// TIA Portal V17 export
// export: Created 2024-08-09T12:53:13.8222628Z, ExportSetting WithDefaults, DisplayName Totally Integrated Automation Portal, DisplayVersion V17 Update 7, DisplayName TIA Portal Openness, DisplayVersion V17 Update 7, DisplayName TIA Portal Version Control Interface, DisplayVersion V17, DisplayName STEP 7 Professional, DisplayVersion V17 Update 7, DisplayName STEP 7 Safety, DisplayVersion V17 Update 6, DisplayName WinCC Professional, DisplayVersion V17 Update 7
VAR_GLOBAL   // PLC tag table "TREMIE_TRAPPE"
END_VAR
VAR_GLOBAL CONSTANT   // user constants
   NIV_TREMIE_TRAPPE_DEBUT_LOT : USInt := 1;
   NIV_TREMIE_TRAPPE_AUT_REMP : USInt := 10;
   NIV_TREMIE_TRAPPE_PRES_PRD : USInt := 20;
   NIV_TREMIE_TRAPPE_ATT_FIN_TROU : USInt := 25;
   NIV_TREMIE_TRAPPE_DEM_EXTRACT : USInt := 30;
   NIV_TREMIE_TRAPPE_NB : USInt := 45;
   NIV_TREMIE_TRAPPE_VID_DEPUIS_X_SEC : USInt := 50;
   NIV_TREMIE_TRAPPE_NIVEAU_BAS : USInt := 60;
   NIV_TREMIE_TRAPPE_TEMPO_MINI : USInt := 70;
   NIV_TREMIE_TRAPPE_DEBUT_VIDANGE : USInt := 90;
   NIV_TREMIE_TRAPPE_FIN_LOT : USInt := 255;
END_VAR
